# EPICS StreamDevice protocol: install/devAPPNAME.proto
ReplyTimeout = 500;
OutTerminator = "\r\n";

@writetimeout { disconnect; }
@replytimeout { disconnect; }
@readtimeout  { disconnect; }
@mismatch     { disconnect; }

getIDN {
    out "PR VR";
    in "%\$1[^\r\n]";
    ExtraInput = Ignore;
}
